Staubli VAL3: loopReadForce.pgx

public program loopReadForce()
begin
  do
    call readForce(nStatus,nForce,nMonitor,bZero,bClear)
    delay(0)
  until (false)
end
